Yaskawa INFORM job: UNSTKING.JBI

/JOB
//NAME UNSTKING
//POS
///NPOS 0,0,0,0,0,0
//INST
///DATE 2025/04/20 21:58
///ATTR SC,RW
///GROUP1 RB1
NOP
'初始化
CALL JOB:STKINIT
'
*LOOP
IFTHENEXP B069=0
	'等待新的数据
	 WAIT B069<>0
ENDIF
'发生异常或者为空时结束
JUMP *LABEL IF B069<>3
'数据复制
CALL JOB:STKCOPY
'一号拆剁位抓取
CALL JOB:UNSTK_PICK01
'一号拆剁位防放置
CALL JOB:UNSTK_PLACE01
*EXIT
END
